FUNCTION_BLOCK FB_Observable_REAL EXTENDS FB_AbstractObservable
VAR
    _fVal:                  REAL;
    _fOldVal:               LREAL;
END_VAR

METHOD FB_init : BOOL
VAR_INPUT
    bInitRetains:       BOOL; // if TRUE, the retain variables are initialized (warm start / cold start)
    bInCopyCode:        BOOL;  // if TRUE, the instance afterwards gets moved into the copy code (online change)
END_VAR
THIS^._nTypeClass := __SYSTEM.TYPE_CLASS.TYPE_REAL;
END_METHOD

PROPERTY fValue32 : REAL
GET
fValue32 := THIS^._fVal;
END_GET
SET
THIS^._fOldVal := _fVal;
THIS^._fVal := fValue32;

THIS^.NotifyWithConditions();
END_SET
END_PROPERTY

PROPERTY nDataSize : UDINT
GET
nDataSize := SIZEOF(REAL);
END_GET
END_PROPERTY

PROPERTY PROTECTED pData : POINTER TO BYTE
GET
pData := ADR(THIS^._fVal);
END_GET
END_PROPERTY

METHOD  ValueChanged : BOOL
VAR_INPUT
END_VAR
ValueChanged := THIS^._fOldVal <> THIS^._fVal;
END_METHOD

END_FUNCTION_BLOCK

(* stored: Version 1.1.0.1, ProductVersion 3.1.4024.12
   POU FB_Observable_REAL: Id {44f2149a-e556-4278-8e29-b5be8430ad03}, SpecialFunc None
   Method FB_init: Id {3358d1bd-7387-03cc-10ee-918907a0ac7e}
   Property fValue32: Id {a0813b3d-f5d1-4dc2-abb7-e188f52cb384}
   Get Get: Id {1b7554b4-9021-4d07-9c73-8d38b15ac4db}
   Set Set: Id {2a2e589f-9528-41d6-9e71-704813bd50f0}
   Property nDataSize: Id {a6262a2d-1b7c-437c-bb14-84a4f343994e}
   Get Get: Id {3d747dd7-b636-4ea4-a95e-ff4ef4c3d281}
   Property pData: Id {a8b5c200-32e8-456f-b91e-3b314a2acf6d}
   Get Get: Id {8d3afe46-0c9f-48a2-9138-5eba426a17a1}
   Method ValueChanged: Id {6e76913e-2d8e-095a-0e47-60a5843d8edb} *)
